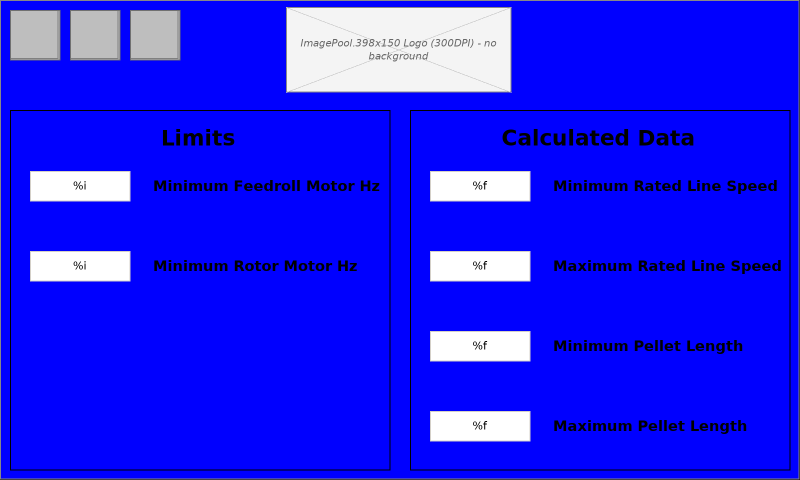
VISUALIZATION Calculations_Settings  // 800x480
    Rectangle (0,0 800x480)
    Rectangle (10,110 380x360)
    Textfield (30,171 100x30), "%i", text variable: GVL.FeedrollMot_Min_Hz
        OnMouseClick: write the text variable via VisuDialogs.Numpad
    Rectangle (410,110 380x360)
    Textfield (30,251 100x30), "%i", text variable: GVL.RotorMot_Min_Hz
        OnMouseClick: write the text variable via VisuDialogs.Keypad
    Textfield (430,411 100x30), "%f", text variable: GVL.Maximum_Pellet_Length
    Image (286,7 225x85), image: ImagePool.398x150 Logo (300DPI) - no background
        OnMouseClick: change screen: Home
    Button (70,10 50x50), image: VisuSymbols.Symbols.Home
        OnMouseClick: change screen: Home
    Label (20,120 357x36), "Limits"
    Label (420,120 357x36), "Calculated Data"
    Button (10,10 50x50), image: VisuSymbols.Symbols.TriangleLeft
        OnMouseClick: change screen: Previous Home
    Textfield (430,171 100x30), "%f", text variable: GVL.Minimum_Line_Speed
    Textfield (430,251 100x30), "%f", text variable: GVL.Maximum_Line_Speed
    Textfield (430,331 100x30), "%f", text variable: GVL.Minimum_Pellet_Length
    Label (150,171 225x30), "Minimum Feedroll Motor Hz"
    Label (150,251 225x30), "Minimum Rotor Motor Hz"
    Label (550,411 225x30), "Maximum Pellet Length"
    Label (550,171 225x30), "Minimum Rated Line Speed"
    Label (550,251 237x30), "Maximum Rated Line Speed"
    Label (550,331 225x30), "Minimum Pellet Length"
    Button (130,10 50x50), image: VisuSymbols.Symbols.TwoWheels
        OnMouseClick: change screen: Settings_Menu
END_VISUALIZATION

(* stored: Version 1.1.0.1, ProductVersion 3.1.4024.12
   Visu Calculations_Settings: Id {77c33add-59ca-4eea-a12a-c44288a64842} *)
